(* IEC 61131-3 sources: 1515t/src, 7 files *)

(* ---- device.st ---- *)
TYPE
    Status : (Stop, Run, Maintain) := Stop;
END_TYPE

INTERFACE Equipment
    METHOD start : BOOL END_METHOD
    METHOD stop : BOOL
        VAR_INPUT

        END_VAR

    END_METHOD

    METHOD getStatus : Status
        VAR_INPUT

        END_VAR
    END_METHOD

END_INTERFACE

CLASS Sensor
    VAR PRIVATE
        sensorId : STRING;
    END_VAR

END_CLASS

(* ---- Class.st ---- *)
CLASS BaseClass
    VAR
        state : INT;    // Available in 'SubClass'
    END_VAR
    VAR PRIVATE
        inner_state : INT;  // Not available in 'SubClass'
    END_VAR
    METHOD Test
        inner_state := 10;
    END_METHOD
    METHOD PRIVATE InnerTest  // Not available in 'SubClass'
        ;
    END_METHOD
END_CLASS

CLASS SubClass EXTENDS BaseClass
    VAR
        additional_state : INT;    // Inherited by 'SubClass'
    END_VAR
    METHOD AdditionalTest
        THIS.Test();    // Access to method of 'BaseClass'
        state := 10;    // Access to fields of 'BaseClass'
        additional_state := 20;
    END_METHOD
END_CLASS

CLASS FINAL SealedSubClass EXTENDS BaseClass
    // 'SealedSubClass' is final and cannot be extended.
END_CLASS

INTERFACE I1
  METHOD MyMethod : INT
      VAR_INPUT
          a : INT := 2;
      END_VAR
  END_METHOD
END_INTERFACE

INTERFACE I2
  METHOD MyMethod : REAL
      VAR_INPUT
          a : REAL := 2;
      END_VAR
  END_METHOD
END_INTERFACE

CLASS MyImplementation IMPLEMENTS I1, I2
    METHOD PUBLIC MyMethod : INT        // Interface methods must be implement as PUBLIC
        VAR_INPUT
            a : INT;
        END_VAR
        VAR_TEMP
            temp : INT;     // You can add temporary variables and code as required.
        END_VAR
        MyMethod := 10;
    END_METHOD

    METHOD PUBLIC MyMethod : REAL        // Interface methods must be implement as PUBLIC
        VAR_INPUT
            a : REAL;
        END_VAR
        VAR_TEMP
            temp : INT;     // You can add temporary variables and code as required.
        END_VAR
        MyMethod := REAL#10.0;
    END_METHOD

    // Error: Class does not implement all interfaces. 'AnotherMethod' is missing.
END_CLASS

CLASS PUBLIC  FINAL A EXTENDS  BaseClass IMPLEMENTS I1, I2
    VAR

    END_VAR
    METHOD PUBLIC MyMethod : INT        // Interface methods must be implement as PUBLIC
        VAR_INPUT
            a : INT;
        END_VAR
        VAR_TEMP
            temp : INT;     // You can add temporary variables and code as required.
        END_VAR
        MyMethod := 10;
    END_METHOD

    METHOD PUBLIC MyMethod : REAL        // Interface methods must be implement as PUBLIC
        VAR_INPUT
            a : REAL;
        END_VAR
        VAR_TEMP
            temp : INT;     // You can add temporary variables and code as required.
        END_VAR
        MyMethod := REAL#10.0;
    END_METHOD

END_CLASS

(* ---- gkc.Geometry.st ---- *)
NAMESPACE gkc.Geometry
    INTERFACE Shape
        METHOD calculateArea : LREAL END_METHOD
    END_INTERFACE

    CLASS ABSTRACT Polygon IMPLEMENTS Shape
        VAR PRIVATE
            sides : int:=3;
        END_VAR
        METHOD PUBLIC ABSTRACT calculateArea : LREAL END_METHOD
        METHOD PUBLIC getSides : Int
            getSides:=sides;
        END_METHOD
        METHOD PUBLIC setSides
            VAR_INPUT
                numberOfSides:int;
            END_VAR
            sides:=numberOfSides;
        END_METHOD
    END_CLASS

    CLASS Triangle EXTENDS Polygon
        VAR PUBLIC
            base : LREAL:=5.0;
            height : LREAL:=10.0;
        END_VAR
        METHOD PUBLIC OVERRIDE calculateArea : LREAL
            calculateArea := base * height / 2;
        END_METHOD
    END_CLASS

    CLASS Square EXTENDS Polygon
        VAR PUBLIC
            sideLength : LREAL:=5.0;
        END_VAR
        METHOD PUBLIC OVERRIDE calculateArea : LREAL
            calculateArea := sideLength * sideLength;
        END_METHOD
    END_CLASS

    CLASS Circle EXTENDS Polygon
        VAR PUBLIC
            radius: LREAL:=5.0;
        END_VAR
        VAR CONSTANT PRIVATE
            PI : LREAL:=3.1415;
        END_VAR
        METHOD PUBLIC OVERRIDE calculateArea : LREAL
            calculateArea:=radius * radius * PI;
        END_METHOD
    END_CLASS
END_NAMESPACE

(* ---- library.st ---- *)
using gkc.math;
NAMESPACE ns1
    class  MyClass
        VAR PRIVATE
            _cal: MyMath;
        END_VAR

        METHOD public Math : Int
            VAR_INPUT
                a : INT;
                b : INT;
                operator : CHAR;

            END_VAR
            VAR_IN_OUT

            END_VAR
            Math:=_cal.Arithmometer(a,b,operator);
        END_METHOD

    END_CLASS
END_NAMESPACE

(* ---- ouc.st ---- *)
USING Siemens.Simatic.S71500.Communication.OUC;

NAMESPACE Tcp

    CLASS OUC
        VAR PRIVATE
            connecting : Connect;
            disconnecting : Disconnect;
            sending : TcpSend;
            receiving : TcpReceive;
        END_VAR
        VAR PUBLIC
            config : ConnectionConfiguration := (Interfaceid := UINT#64, RemoteAddress := [BYTE#192, BYTE#168, BYTE#200, BYTE#19]);
            connected : BOOL;
        END_VAR

        METHOD PUBLIC connect : BOOL
            VAR_OUTPUT
                error : BOOL;
                status : WORD;
            END_VAR
            connecting(execute := NOT connected AND NOT connecting.busy, connectionID := config.ConnectionID, connectionConfiguration := config, status => status, error => error);
            IF connecting.done THEN
                connected := TRUE;
            END_IF;
            connect := connected;
        END_METHOD

        METHOD PUBLIC disconnect
            VAR_INPUT
                execute : BOOL;
            END_VAR
            disconnecting(execute := connected AND NOT disconnecting.busy AND execute, connectionID := config.ConnectionID);
            IF disconnecting.done THEN
                connected := FALSE;
            END_IF;
        END_METHOD

        METHOD PUBLIC send
            VAR_INPUT
                req : BOOL;
                length : UDINT := UDINT#5;
            END_VAR
            VAR_IN_OUT
                data : ARRAY[*] OF BYTE;
            END_VAR
            VAR_OUTPUT
                done : BOOL;
                error : BOOL;
            END_VAR
            sending(execute := connected AND req, connectionID := config.ConnectionID, length := UDINT#5, data := data, done => done, error => error);
        END_METHOD

        METHOD PUBLIC receive
            VAR_IN_OUT
                data : ARRAY[*] OF BYTE;
            END_VAR
            receiving(enable := connected, connectionID := config.ConnectionID, adhocMode := TRUE, data := data);
        END_METHOD
    END_CLASS

END_NAMESPACE

(* ---- configuration.st ---- *)
USING Siemens.Simatic.S71500.Tasks;
CONFIGURATION MyConfiguration
    TASK Main(Priority := 1, INTERVAL:=t#100ms);

    PROGRAM P1 WITH Main: MainProgram;
    {S7.extern=ReadWrite}
    {OpcUa.AccessLevel = ReadWrite}
    VAR_GLOBAL
        ET200SP_DI1_InputAddress AT %IB0: BYTE;
        {OpcUa.AccessLevel = ReadOnly}
        ET200SP_DQ1_OutputAddress AT %QB2: BYTE;
        // {OpcUa.AccessLevel = Hidden}
        sinData,cosData : REAL;
        AI1_CH0 AT %IW1: WORD;
        AI1_CH1 AT %IW3: WORD;

    // END_VAR
    // VAR_GLOBAL
        count: LREAL:= 0.0;
        temperature: REAL;
        result:int;
    END_VAR
END_CONFIGURATION

(* ---- MainProgram.st ---- *)
USING Siemens.Simatic.S71500.Clocks;
USING System.DateTime;
USING System.FastMath;

PROGRAM  MainProgram
    VAR_EXTERNAL
        ET200SP_DQ1_OutputAddress:BYTE;
        sinData,cosData  : REAL;
        count:LREAL ;
        AI1_CH0  : WORD;
        AI1_CH1  : WORD;
        temperature: REAL;
        result:int;

    END_VAR
    VAR_INPUT
        // cal:ns1.MyClass;
    END_VAR
    VAR_OUTPUT
    END_VAR
    VAR_IN_OUT

    END_VAR
    VAR
        cal:ns1.MyClass;
    END_VAR
    VAR_TEMP
        systemDateTime : LDATE_AND_TIME;
        year, month, day, second ,millisecond: INT;
    END_VAR
    ET200SP_DQ1_OutputAddress := ET200SP_DQ1_OutputAddress XOR BYTE#01 ;
    // GetSystemDateTime(value => systemDateTime);
    // SplitDateAndTime(
    //     value := systemDateTime,
    //     millisecond => millisecond
    // );
    count := count + 0.01 ;
    sinData := sin(TO_REAL( count));
    cosData := cos(TO_REAL( count));
    temperature:=TO_REAL(TO_INT (AI1_CH0)) / TO_REAL( 276.48);
    result:=cal.Math(TO_INT (count),1,'+');

END_PROGRAM
